PROGRAM P_Demo_FB_DALIV2RecallMaxLevel
VAR
    fbFB_DALIV2RecallMaxLevel        : FB_DALIV2RecallMaxLevel;
    stCommandBuffer : ST_DALIV2CommandBuffer;

    bTrigger        : BOOL;
    nLampAddr        : BYTE := 0;


    bBusy           : BOOL;
    bErr            : BOOL;
    nErrId          : UDINT;
END_VAR

// =============================================================================
// 场景：应急联动：火警触发，PLC 广播本 FB 给所有应急灯，自动全亮（按 `MAX VALUE` 配置，通常 254）。...
//
// 价值：DALI 协议标准命令的轻量封装。
//
// 验证步骤：
//   1. 通信 FB 跑起；编译；登录。
//   2. 在线 bTrigger 一次上升沿；等 bBusy 回 FALSE。
//   3. 观察 short addr 0 灯的物理亮度变化是否符合本命令描述。
// =============================================================================
fbFB_DALIV2RecallMaxLevel(
    bStart           := bTrigger,
    nAddr            := nLampAddr,
    eAddrType        := eDALIV2AddrTypeShort,
    eCommandPriority := eDALIV2CommandPriorityMiddle,
    stCommandBuffer  := stCommandBuffer
);

bBusy  := fbFB_DALIV2RecallMaxLevel.bBusy;
bErr   := fbFB_DALIV2RecallMaxLevel.bError;
nErrId := fbFB_DALIV2RecallMaxLevel.nErrorId;

END_PROGRAM

(* stored: Version 1.1.0.1, ProductVersion 3.1.4024.5
   POU P_Demo_FB_DALIV2RecallMaxLevel: Id {a063602d-6e18-5007-abe9-777967777fc7}, SpecialFunc None *)
